/// Fast Task program
PROGRAM P_Fast
VAR CONSTANT
	iMaxTaskAllocation				: INT := 10;
END_VAR

VAR
	ii	: INT;
	aItfTasks						: ARRAY[0..255] OF ITF_TaskAllocation;	  
END_VAR

/// run cyclic fast tasks
FOR ii := 0 TO iMaxTaskAllocation DO
	IF aItfTasks[ii] = 0 THEN
		CONTINUE;
	END_IF
	IF aItfTasks[ii].Task = E_Task.eTask_fast THEN
		aItfTasks[ii].Invoke();
	END_IF
END_FOR

METHOD RegisterTask : E_OperationResult
VAR_INPUT
	/// Task to be registered
	ITask	: ITF_TaskAllocation;
END_VAR
VAR
	ii	: INT;
END_VAR
/// queue task
FOR ii := 0 TO iMaxTaskAllocation DO
	IF aItfTasks[ii] <> 0 THEN
		IF aItfTasks[ii].TaskId <> ITask.TaskId THEN
			CONTINUE;
		END_IF
	END_IF
	ITask.TaskId := ii + 1;
	aItfTasks[ii] := ITask;
	EXIT;
END_FOR
END_METHOD

METHOD UnregisterTask : E_OperationResult
VAR_INPUT
	/// Task to be unregistered
	ITask	: ITF_TaskAllocation;
END_VAR
VAR
	ii	: INT;
END_VAR
/// dequeue task
FOR ii := 0 TO iMaxTaskAllocation DO
	IF aItfTasks[ii] = 0 THEN
		CONTINUE;
	END_IF
	IF aItfTasks[ii].TaskId <> ITask.TaskId THEN
		CONTINUE;
	END_IF
	aItfTasks[ii] := 0;
END_FOR
END_METHOD

END_PROGRAM

(* stored: Version 1.1.0.1, ProductVersion 3.1.4022.9
   POU P_Fast: Id {7047c25d-a1ce-442b-b871-40c96cfb03bb}, SpecialFunc None
   Method RegisterTask: Id {f9918118-ef6a-461d-bcb4-e5063c741d59}
   Method UnregisterTask: Id {c7ea2e1a-97e0-4923-8c7a-d8f1ccd94c79} *)
